FUNCTION_BLOCK FB_EMERGENCY_SYS
VAR_IN_OUT
	stSystem: sysType;         // ALLOW CHILD METHODS TO ACCESS DATA
END_VAR


CASE stSystem.state OF

    // ==========================================
    // INITIAL STATES
    // ==========================================
    sysState.stDisconnected:
        IF stSystem.transitions.T1 THEN
            stSystem.state := sysState.stClosing;
        END_IF

    sysState.stOpening:
        IF stSystem.transitions.T2 THEN
            stSystem.state := sysState.stDisconnected;
        END_IF

    sysState.stClosing:
        IF stSystem.transitions.T3 THEN
            stSystem.state := sysState.stWaitingRaspberry;
        END_IF

    // ==========================================
    // WAIT AND RASPBERRY CONNECTION
    // ==========================================
    sysState.stWaitingRaspberry:
        IF stSystem.transitions.T4 THEN
            stSystem.state := sysState.stOpening;
        ELSIF stSystem.transitions.T7 THEN
            stSystem.state := sysState.stAlarmOpening;
        ELSIF stSystem.transitions.T8 THEN
            stSystem.state := sysState.stFaceDetectionAlarmOpening;
        ELSIF stSystem.transitions.T9 THEN
            stSystem.state := sysState.stConfigOpening;
        ELSIF stSystem.transitions.T5 THEN
            stSystem.state := sysState.stRaspberryFailOpening;
        ELSIF stSystem.transitions.T6 THEN
            stSystem.state := sysState.stRaspberryOk;
        END_IF

    sysState.stRaspberryOk:
        IF stSystem.transitions.T10 THEN
            stSystem.state := sysState.stOpening;
        ELSIF stSystem.transitions.T12 THEN
            stSystem.state := sysState.stAlarmOpening;
        ELSIF stSystem.transitions.T13 THEN
            stSystem.state := sysState.stFaceDetectionAlarmOpening;
        ELSIF stSystem.transitions.T14 THEN
            stSystem.state := sysState.stConfigOpening;
        ELSIF stSystem.transitions.T11 THEN
            stSystem.state := sysState.stWaitingRaspberry;
        END_IF

    // ==========================================
    // DEFAULT ALARM
    // ==========================================
    sysState.stAlarmOpening:
        IF stSystem.transitions.T15 THEN
            stSystem.state := sysState.stAlarm;
        END_IF

    sysState.stAlarm:
        IF stSystem.transitions.T16 THEN
            stSystem.state := sysState.stAlarmClosing;
        END_IF

    sysState.stAlarmClosing:
        IF stSystem.transitions.T17 THEN
            stSystem.state := sysState.stWaitingRaspberry;
        END_IF

    // ==========================================
    // FACIAL DETECTION ALARM
    // ==========================================
    sysState.stFaceDetectionAlarmOpening:
        IF stSystem.transitions.T18 THEN
            stSystem.state := sysState.stFaceDetectionAlarm;
        END_IF

    sysState.stFaceDetectionAlarm:
        IF stSystem.transitions.T19 THEN
            stSystem.state := sysState.stFaceDetectionAlarmClosing;
        END_IF

    sysState.stFaceDetectionAlarmClosing:
        IF stSystem.transitions.T20 THEN
            stSystem.state := sysState.stWaitingRaspberry;
        END_IF

    // ==========================================
    // TEST MODE
    // ==========================================
    sysState.stConfigOpening:
        IF stSystem.transitions.T21 THEN
            stSystem.state := sysState.stConfig;
        END_IF

    sysState.stConfig:
        IF stSystem.transitions.T22 THEN
            stSystem.state := sysState.stConfigClosing;
        END_IF

    sysState.stConfigClosing:
        IF stSystem.transitions.T23 THEN
            stSystem.state := sysState.stWaitingRaspberry;
        END_IF

    // ==========================================
    // RASPBERRY PI ERROR
    // ==========================================
    sysState.stRaspberryFailOpening:
        IF stSystem.transitions.T24 THEN
            stSystem.state := sysState.stRaspberryFail;
        END_IF

    sysState.stRaspberryFail:
        IF stSystem.transitions.T25 THEN
            stSystem.state := sysState.stDisconnected;
        END_IF

END_CASE

METHOD mOutputs
VAR_IN_OUT
    stSystem: sysType;
END_VAR
// ==============================================================================
// Method: mOutputs
// Description: Triggers corresponding outputs in each state
// ==============================================================================

stSystem.outputs.oOpenDoor :=
    (stSystem.state = sysState.stOpening) OR
    (stSystem.state = sysState.stAlarmOpening) OR
    (stSystem.state = sysState.stFaceDetectionAlarmOpening) OR
    (stSystem.state = sysState.stConfigOpening) OR
    (stSystem.state = sysState.stRaspberryFailOpening);

// --- oCloseDoor: active in all Closing states ---
stSystem.outputs.oCloseDoor :=
    (stSystem.state = sysState.stClosing) OR
    (stSystem.state = sysState.stAlarmClosing) OR
    (stSystem.state = sysState.stFaceDetectionAlarmClosing) OR
    (stSystem.state = sysState.stConfigClosing);

// --- oAlarm: active during any alarm state (both alarm types, all sub-states) ---
stSystem.outputs.oAlarm :=
    (stSystem.state = sysState.stAlarmOpening) OR
    (stSystem.state = sysState.stAlarm) OR
    (stSystem.state = sysState.stAlarmClosing) OR
    (stSystem.state = sysState.stFaceDetectionAlarmOpening) OR
    (stSystem.state = sysState.stFaceDetectionAlarm) OR
    (stSystem.state = sysState.stFaceDetectionAlarmClosing) OR
(stSystem.state = sysState.stRaspberryFailOpening) OR
(stSystem.state = sysState.stRaspberryFail);
END_METHOD

METHOD mTransitions : BOOL
VAR_IN_OUT
    stSystem: sysType;
	
	
END_VAR
// ==============================================================================
// Method: mTransitions
// Description: Evaluates and triggers the boolean flags for state transitions
//              based on the current state and specific logical conditions.
// ==============================================================================

stSystem.inputs.iReedSwitch_rtrig(CLK := stSystem.inputs.iReedSwitch); // Define R_TRIG CLK for Reed Switch

// Transition T1: FROM stDisconnected TO stClosing WHEN iSwitch is TRUE
stSystem.transitions.T1 := (stSystem.state = sysState.stDisconnected) AND (stSystem.inputs.iSwitch = TRUE);

// Transition T2: FROM stOpening TO stDisconnected WHEN doorOpenTimer is done
stSystem.transitions.T2 := (stSystem.state = sysState.stOpening) AND (stSystem.inputs.iReedSwitch_rtrig.Q = TRUE);

// Transition T3: FROM stClosing TO stWaitingRaspberry WHEN doorCloseTimer is done
stSystem.transitions.T3 := (stSystem.state = sysState.stClosing) AND (stSystem.inputs.iReedSwitch_rtrig.Q = TRUE);

// Transition T4: FROM stWaitingRaspberry TO stOpening WHEN iSwitch is FALSE
stSystem.transitions.T4 := (stSystem.state = sysState.stWaitingRaspberry) AND (stSystem.inputs.iSwitch = FALSE);

// ... you must continue this pattern up to T25 following the transition table.

// T5: FROM stWaitingRaspberry TO stRaspberryFailOpening WHEN rpiWaitTimer done
stSystem.transitions.T5 := (stSystem.state = sysState.stWaitingRaspberry) AND (stSystem.timersCounters.rpiWaitTimer.Q = TRUE);

// T6: FROM stWaitingRaspberry TO stRaspberryOk WHEN RPi pong received
stSystem.transitions.T6 := (stSystem.state = sysState.stWaitingRaspberry) AND (stSystem.RpiWatchdog.iRPiFail = FALSE);

// T7: FROM stWaitingRaspberry TO stAlarmOpening WHEN alarm button pressed
stSystem.transitions.T7 := (stSystem.state = sysState.stWaitingRaspberry) AND (stSystem.inputs.iAlarmButton = FALSE);

// T8: FROM stWaitingRaspberry TO stFaceDetectionAlarmOpening WHEN face detected
stSystem.transitions.T8 := (stSystem.state = sysState.stWaitingRaspberry) AND (stSystem.inputs.iFacialDetec = TRUE);
 	
// T9: FROM stWaitingRaspberry TO stConfigOpening WHEN test button pressed
stSystem.transitions.T9 := (stSystem.state = sysState.stWaitingRaspberry) AND (stSystem.inputs.iTestButton = TRUE);

// T10: FROM stRaspberryOk TO stOpening WHEN iSwitch is FALSE
stSystem.transitions.T10 := (stSystem.state = sysState.stRaspberryOk) AND (stSystem.inputs.iSwitch = FALSE);

// T11: FROM stRaspberryOk TO stWaitingRaspberry WHEN rpiPingTimer done
stSystem.transitions.T11 := (stSystem.state = sysState.stRaspberryOk) AND (stSystem.timersCounters.rpiPingTimer.Q = TRUE);

// T12: FROM stRaspberryOk TO stAlarmOpening WHEN alarm button pressed
stSystem.transitions.T12 := (stSystem.state = sysState.stRaspberryOk) AND (stSystem.inputs.iAlarmButton = FALSE);

// T13: FROM stRaspberryOk TO stFaceDetectionAlarmOpening WHEN face detected
stSystem.transitions.T13 := (stSystem.state = sysState.stRaspberryOk) AND (stSystem.inputs.iFacialDetec = TRUE);

// T14: FROM stRaspberryOk TO stConfigOpening WHEN test button pressed
stSystem.transitions.T14 := (stSystem.state = sysState.stRaspberryOk) AND (stSystem.inputs.iTestButton = TRUE);

// T15: FROM stAlarmOpening TO stAlarm WHEN doorOpenTimer done
stSystem.transitions.T15 := (stSystem.state = sysState.stAlarmOpening) AND (stSystem.inputs.iReedSwitch_rtrig.Q = TRUE);

// T16: FROM stAlarm TO stAlarmClosing WHEN test button AND alarm cleared
stSystem.transitions.T16 := (stSystem.state = sysState.stAlarm) AND (stSystem.inputs.iTestButton = TRUE) AND (stSystem.inputs.iAlarmButton = FALSE);

// T17: FROM stAlarmClosing TO stWaitingRaspberry WHEN doorCloseTimer done
stSystem.transitions.T17 := (stSystem.state = sysState.stAlarmClosing) AND (stSystem.inputs.iReedSwitch_rtrig.Q = TRUE);

// T18: FROM stFaceDetectionAlarmOpening TO stFaceDetectionAlarm WHEN doorOpenTimer done
stSystem.transitions.T18 := (stSystem.state = sysState.stFaceDetectionAlarmOpening) AND (stSystem.inputs.iReedSwitch_rtrig.Q = TRUE);

// T19: FROM stFaceDetectionAlarm TO stFaceDetectionAlarmClosing WHEN test button AND alarm cleared
stSystem.transitions.T19 := (stSystem.state = sysState.stFaceDetectionAlarm) AND (stSystem.inputs.iTestButton = TRUE) AND (stSystem.inputs.iAlarmButton = FALSE);

// T20: FROM stFaceDetectionAlarmClosing TO stWaitingRaspberry WHEN doorCloseTimer done
stSystem.transitions.T20 := (stSystem.state = sysState.stFaceDetectionAlarmClosing) AND (stSystem.inputs.iReedSwitch_rtrig.Q = TRUE);

// T21: FROM stConfigOpening TO stConfig WHEN doorOpenTimer done
stSystem.transitions.T21 := (stSystem.state = sysState.stConfigOpening) AND (stSystem.inputs.iReedSwitch_rtrig.Q = TRUE);

// T22: FROM stConfig TO stConfigClosing WHEN test button pressed
stSystem.transitions.T22 := (stSystem.state = sysState.stConfig) AND (stSystem.inputs.iTestButton = TRUE);

// T23: FROM stConfigClosing TO stWaitingRaspberry WHEN doorCloseTimer done
stSystem.transitions.T23 := (stSystem.state = sysState.stConfigClosing) AND (stSystem.inputs.iReedSwitch_rtrig.Q = TRUE);

// T24: FROM stRaspberryFailOpening TO stRaspberryFail WHEN doorOpenTimer done
stSystem.transitions.T24 := (stSystem.state = sysState.stRaspberryFailOpening) AND (stSystem.inputs.iReedSwitch_rtrig.Q = TRUE);

// T25: FROM stRaspberryFail TO stDisconnected WHEN iSwitch is FALSE
stSystem.transitions.T25 := (stSystem.state = sysState.stRaspberryFail) AND (stSystem.inputs.iSwitch = FALSE);

// T26: FROM stAlarmClosing TO stAlarmOpening WHEN alarm button pressed
stSystem.transitions.T26 := (stSystem.state = sysState.stAlarmClosing) AND (stSystem.inputs.iAlarmButton = FALSE);

// T27: FROM stAlarmClosing TO stFaceDetectionAlarmOpening WHEN face detected
stSystem.transitions.T27 := (stSystem.state = sysState.stAlarmClosing) AND (stSystem.inputs.iFacialDetec = TRUE);

// T28: FROM stAlarmClosing TO stConfigOpening WHEN test button pressed
stSystem.transitions.T28 := (stSystem.state = sysState.stAlarmClosing) AND (stSystem.inputs.iTestButton = TRUE);

// T29: FROM stFaceDetectionAlarmClosing TO stAlarmOpening WHEN alarm button pressed
stSystem.transitions.T29 := (stSystem.state = sysState.stFaceDetectionAlarmClosing) AND (stSystem.inputs.iAlarmButton = FALSE);

// T30: FROM stFaceDetectionAlarmClosing TO stFaceDetectionAlarmOpening WHEN face detected
stSystem.transitions.T30 := (stSystem.state = sysState.stFaceDetectionAlarmClosing) AND (stSystem.inputs.iFacialDetec = TRUE);

// T31: FROM stFaceDetectionAlarmClosing TO stConfigOpening WHEN test button pressed
stSystem.transitions.T31 := (stSystem.state = sysState.stFaceDetectionAlarmClosing) AND (stSystem.inputs.iTestButton = TRUE);

// T32: FROM stConfigClosing TO stAlarmOpening WHEN alarm button pressed
stSystem.transitions.T32 := (stSystem.state = sysState.stConfigClosing) AND (stSystem.inputs.iAlarmButton = FALSE);

// T33: FROM stConfigClosing TO stFaceDetectionAlarmOpening WHEN face detected
stSystem.transitions.T33 := (stSystem.state = sysState.stConfigClosing) AND (stSystem.inputs.iFacialDetec = TRUE);

// T34: FROM stConfigClosing TO stConfigOpening WHEN test button pressed
stSystem.transitions.T34 := (stSystem.state = sysState.stConfigClosing) AND (stSystem.inputs.iTestButton = TRUE);

// T35: FROM stFaceDetectionAlarmOpening TO stFaceDetectionAlarmClosing WHEN test button AND alarm cleared
stSystem.transitions.T35 := (stSystem.state = sysState.stFaceDetectionAlarmOpening) AND (stSystem.inputs.iTestButton = TRUE) AND (stSystem.inputs.iAlarmButton = FALSE);

// T36: FROM stConfigOpening TO stConfigClosing WHEN test button AND alarm cleared
stSystem.transitions.T36 := (stSystem.state = sysState.stConfigOpening) AND (stSystem.inputs.iTestButton = TRUE) AND (stSystem.inputs.iAlarmButton = FALSE);

// T37: FROM stAlarmOpening TO stAlarmClosing WHEN test button AND alarm cleared
stSystem.transitions.T37 := (stSystem.state = sysState.stAlarmOpening) AND (stSystem.inputs.iTestButton = TRUE) AND (stSystem.inputs.iAlarmButton = FALSE);
END_METHOD

END_FUNCTION_BLOCK

(* stored: Version 1.1.0.1, ProductVersion 3.1.4026.18
   POU FB_EMERGENCY_SYS: Id {037855c0-4683-4fd0-aa20-772e94d3b895}, SpecialFunc None
   Method mOutputs: Id {83f6b582-9dbd-4b31-83b6-b11bcde56274}
   Method mTransitions: Id {1b7dd8b6-9891-4637-828c-17df8373d614} *)
